(* PLC project OOP_Curso, Beckhoff Automation GmbH TwinCAT PLC Control 3.5.13.21 *)
(* stored: creationDateTime 2023-08-07T09:41:19.4338283, modificationDateTime 2023-08-07T09:41:19.4377308 *)

FUNCTION_BLOCK FB_Coche EXTENDS FB_Vehiculo
VAR_INPUT
	velocidadMaxima : REAL;
END_VAR
VAR_OUTPUT
END_VAR
VAR
END_VAR

            
          

METHOD getVelocidadMaxima : REAL
VAR_INPUT
END_VAR
                  getVelocidadMaxima := velocidadMaxima;
                
END_METHOD
END_FUNCTION_BLOCK

FUNCTION_BLOCK FB_Moto EXTENDS FB_Vehiculo
VAR_INPUT
	aceleracion : REAL;
END_VAR
VAR_OUTPUT
END_VAR
VAR
END_VAR

            
          

METHOD getAceleracion : REAL
VAR_INPUT
END_VAR
                  getAceleracion := aceleracion;
                
END_METHOD
END_FUNCTION_BLOCK

FUNCTION_BLOCK FB_Vehiculo
VAR_INPUT
	velocidad : REAL;
END_VAR
VAR_OUTPUT
END_VAR
VAR
END_VAR

            
          

METHOD getVelocidad : REAL
VAR_INPUT
END_VAR
                  getVelocidad := velocidad;
                
END_METHOD
END_FUNCTION_BLOCK

PROGRAM _25_SOLID_OCP
VAR
	Audi_A8 : FB_Coche;
	Audi_A8_Velocidad :REAL;
	Audi_A8_VelocidadMaxima : REAL;
	
	Suzuki_Ninja : FB_Moto;
	Suzuki_Ninja_Velocidad :REAL;
	Suzuki_Ninja_Aceleracion :REAL;
END_VAR

            //Llamada al objeto Audi_A8.
Audi_A8();
//Este metodo es heredado de la clase Vehiculo.
Audi_A8_Velocidad := Audi_A8.getVelocidad(); 
//Este método es propio de la clase Coche.
Audi_A8_VelocidadMaxima := Audi_A8.getVelocidadMaxima();

//Llamada al objeto Suzuki Ninja.
Suzuki_Ninja();
//Este metodo es heredado de la clase Vehiculo
Suzuki_Ninja_Velocidad := Suzuki_Ninja.getVelocidad();
//Este método es propio de la clase Moto.
Suzuki_Ninja_Aceleracion := Suzuki_Ninja.getAceleracion();
          
END_PROGRAM
